PROGRAM MAIN
VAR
END_VAR

COM_DataMaster();
COM_DataSlave();

END_PROGRAM

(* stored: Version 1.1.0.1, ProductVersion 3.1.4022.18
   POU MAIN: Id {fe563e4f-7aeb-4f3e-9b34-419720cc2af3}, SpecialFunc None *)
